FUNCTION_BLOCK FB_BaseComponentDecoratorParent EXTENDS FB_BaseLoggerElementDecoratorParent IMPLEMENTS ITF_BaseComponentDecoratorParent
VAR
	itfComponent				: ITF_BaseComponent;
END_VAR

(*			
	EVERDE sp. z o.o.
	Rafał Osajda		27.03.2025		TC 4024.66
	Obsluga bledow sprawdzanie czy jakis blad sie nei pojawil i ustawienie stanu lub wylaczenie
*)
METHOD PUBLIC ExecuteEveryCycle_Error
VAR_INPUT
END_VAR
THIS^.itfComponent.ExecuteEveryCycle_Error ();
END_METHOD

(*			
	EVERDE sp. z o.o.
	Rafał Osajda		27.03.2025		TC 4024.66
	Wywolanie co cykl operacji 
*)
METHOD PUBLIC ExecuteEveryCycle_Operation
VAR_INPUT
END_VAR
THIS^.ExecuteEveryCycle_Operation ();
END_METHOD

(*			
	EVERDE sp. z o.o.
	Rafał Osajda		27.03.2025		TC 4024.66
	Aktualizacja flag 
*)
METHOD PUBLIC ExecuteEveryCycle_Status
VAR_INST
END_VAR
THIS^.ExecuteEveryCycle_Status ();
END_METHOD

(*			
	EVERDE sp. z o.o.
	Rafał Osajda		27.03.2025		TC 4024.66
	Testowanie czy nei pojawil sie jakis rozkaz i uruchomienie odpowiednich operacji
*)
METHOD PUBLIC ExecuteEveryCycle_Test
VAR_INPUT
END_VAR
THIS^.ExecuteEveryCycle_Test ();
END_METHOD

(*			
	EVERDE sp. z o.o.
	Rafał Osajda		03.10.2025		TC 4024.66
	
*)
METHOD PUBLIC FirstCycle : BOOL
VAR_INPUT
END_VAR
FirstCycle				:= THIS^.FirstCycle ();
END_METHOD

(*			
	EVERDE sp. z o.o.
	Rafał Osajda		07.10.2025		TC 4024.66
	Dodpisywanie się do listy logera
*)
METHOD PUBLIC JoinTheLogger : BOOL
VAR_INPUT
END_VAR
JoinTheLogger	:= THIS^.itfComponent.JoinTheLogger ();
END_METHOD

METHOD PUBLIC Reset : BOOL
VAR_INPUT
END_VAR
Reset	:= THIS^.itfComponent.Reset ();
END_METHOD

METHOD PUBLIC ResetGetBusy : BOOL
VAR_INPUT
END_VAR
ResetGetBusy		:= THIS^.itfComponent.ResetGetBusy ();
END_METHOD

METHOD PUBLIC ResetGetStatus : BOOL
VAR_INPUT
END_VAR
ResetGetStatus			:= THIS^.itfComponent.ResetGetStatus ();
END_METHOD

END_FUNCTION_BLOCK

(* stored: Version 1.1.0.1, ProductVersion 3.1.4024.15
   POU FB_BaseComponentDecoratorParent: Id {d301a0ba-63d7-4941-8c82-98d9202ac34c}, SpecialFunc None
   Folder ITF_BaseComponent: Id {c1425345-0a97-4881-9b46-35bd773e4177}
   Method ExecuteEveryCycle_Error: Id {a0d49fb3-4440-46c8-b692-5a69fa9df254}
   Method ExecuteEveryCycle_Operation: Id {211c994c-be49-4417-9223-2155aabf14dc}
   Method ExecuteEveryCycle_Status: Id {323c175a-7a7a-40de-9e52-6b8cb429aaed}
   Method ExecuteEveryCycle_Test: Id {311c07d1-160a-4b1e-a1b1-725afc5a0e4b}
   Method FirstCycle: Id {29fba4ac-b428-4421-8774-7f28cfa81e67}
   Method JoinTheLogger: Id {b346dd79-7a2a-4783-8d62-c868aaa6ec7b}
   Method Reset: Id {b09281d3-70a6-481f-97cd-584f5bd951d5}
   Method ResetGetBusy: Id {4ba919e7-fd9d-4960-b107-79433ddc9ae9}
   Method ResetGetStatus: Id {a84ce79a-b00e-41d5-b194-94c769ff7b31} *)
